TYPE MoverSequenceInfo :
STRUCT
	MoverId : UDINT;
	CurrentStation : INT;
	Velocity : MC_LREAL;
	State : IndexSequenceState;
END_STRUCT
END_TYPE

(* stored: Version 1.1.0.1, ProductVersion 3.1.4024.12
   DUT MoverSequenceInfo: Id {e31e4eaf-6c71-46bd-8e49-86316a781b98} *)
